{attribute 'qualified_only'}
VAR_GLOBAL
	
	database: ARRAY[0..MAX_CSV_ROWS, 0..MAX_CSV_COLUMNS] OF STRING;
	
	dataArray: ARRAY[0..MAX_CSV_ROWS, 0..MAX_CSV_COLUMNS] OF STRING;
END_VAR

VAR_GLOBAL CONSTANT
	MAX_CSV_COLUMNS			:INT:=99;
	MAX_CSV_ROWS			: INT:=99;
END_VAR

(* stored: Version 1.1.0.1, ProductVersion 3.1.4022.16
   GVL GVL_General: Id {1b3fd15b-5b52-4df0-ba52-42c3fdfcd81c} *)
